FUNCTION_BLOCK FlipFlop (* Composite Function Block Type *)
  (* Standard: 61499-2 *)
  (* Version 0.0, 2014-04-28, 4DIAC-IDE, 4DIAC-Consortium *)
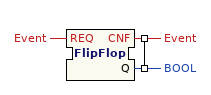
  EVENT_INPUT
    REQ; (* Trigger FlipFlop *)
  END_EVENT
  EVENT_OUTPUT
    CNF WITH Q; (* Event Out *)
  END_EVENT
  VAR_OUTPUT
    Q : BOOL; (* Output value *)
  END_VAR
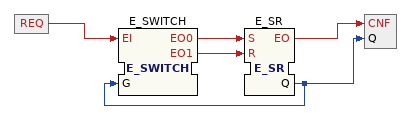
  FBS
    E_SR : E_SR;
    E_SWITCH : E_SWITCH;
  END_FBS
  EVENT_CONNECTIONS
    E_SWITCH.EO0 TO E_SR.S;
    E_SWITCH.EO1 TO E_SR.R;
    E_SR.EO TO CNF;
    REQ TO E_SWITCH.EI;
  END_CONNECTIONS
  DATA_CONNECTIONS
    E_SR.Q TO Q;
    E_SR.Q TO E_SWITCH.G;
  END_CONNECTIONS
END_FUNCTION_BLOCK
